Universal Robots PolyScope program: kg_client.urp

Program kg_client (installation=default directory=/home/kieran/ursim-3.12.1.90940/programs createdIn=3.3.4.310 lastSavedIn=3.12.1.90940 robotSerialNumber=2018359999)
Calibrated DH parameters: a=[0.00011, -0.28299, -0.391817, -0.000036, 0.000148, 0]; d=[0.089132, -365.338436, 366.566923, -1.118136, 0.094823, 0.082571]; alpha=[1.570367, -0.000867, -0.014051, 1.570127, -1.570349, 0]; deltaTheta=[0.000049, 0.840298, -0.88576, 0.044111, 0.000904, -0.000211]
BeforeStart
  var_1 := False
  thread_flag := False
  var_10 := [0,0,0,0,0,0,0,0,0,0]
  Set NoAction tcp=TCP
Robot Program (runOnlyOnce=false)
  Loop While (checkContinuously=false) expression=var_1==False
    var_1 := socket_open("127.0.0.1",30010)
    Wait Sleep waitTime=0.5
  Loop While (checkContinuously=true) expression=var_1== True
    Wait Sleep waitTime=0.001
    var_2 := socket_read_ascii_float(12)
    Loop While (checkContinuously=false) expression=var_2[0]≠12
      var_2 := socket_read_ascii_float(12)
    Switch expression=var_2[1]
      Case (caseValue=0)
        'movejl'
        var_3 := p[var_2[2],var_2[3],var_2[4],var_2[5],var_2[6],var_2[7]]
        Script: movej(var_3,var_2[8],var_2[9],var_2[10],var_2[11])
        If var_2[12]==0
          Script: socket_send_string("completed_pose_move")
      Case (caseValue=1)
        'movej'
        var_6 := [var_2[2],var_2[3],var_2[4],var_2[5],var_2[6],var_2[7]]
        Script: movej(var_6,var_2[8],var_2[9],var_2[10],var_2[11])
        If var_2[12]==0
          Script: socket_send_string("completed_joint_move")
      Case (caseValue=2)
        'movel'
        var_3 := p[var_2[2],var_2[3],var_2[4],var_2[5],var_2[6],var_2[7]]
        Script: movel(var_3,var_2[8],var_2[9],var_2[10],var_2[11])
        If var_2[12]==0
          Script: socket_send_string("completed_linear_move")
      Case (caseValue=3)
        'move to var_3 relative to current pose'
        var_3 := p[var_2[2],var_2[3],var_2[4],var_2[5],var_2[6],var_2[7]]
        var_5 := get_actual_tcp_pose()
        Script: movel(pose_trans(var_5,var_3),var_2[8],var_2[9],var_2[10],var_2[11])
        If var_2[12]==0
          Script: socket_send_string("completed_relative_linear_move")
      Case (caseValue=4)
        'force move in single axis'
        var_5 := get_actual_tcp_pose()
        If var_2[2]≠0
          Script: var_5[0]=var_5[0]+var_2[2]
          axis := 0
        ElseIf var_2[3]≠0
          Script: var_5[1]=var_5[1]+var_2[3]
          axis := 1
        ElseIf var_2[4]≠0
          Script: var_5[2]=var_5[2]+var_2[4]
          axis := 2
        Script: thread_flag= True
        Loop While (checkContinuously=true) expression=thread_flag== True
          Script: movel(var_5,var_2[8],var_2[9],0,0)
          Wait Sleep waitTime=0.01
          Script: thread_flag= False
        Script: stopl(10)
        If var_2[12]==0
          Script: socket_send_string("completed_force_move")
      Case (caseValue=5)
        'servoj'
        var_3 := p[var_2[2],var_2[3],var_2[4],var_2[5],var_2[6],var_2[7]]
        If var_2[12]==0
          Script: stopl(0.5)
        Else 
          var_14 := get_inverse_kin(var_3)
          Script: servoj(var_14,t=var_2[9],lookahead_time=var_2[10],gain=var_2[11])
        If var_2[12]==0
          Script: socket_send_string("completed_servoj_move")
      Case (caseValue=6)
        'speedl'
        var_6 := [var_2[2],var_2[3],var_2[4],var_2[5],var_2[6],var_2[7]]
        If var_2[10]==0
          Script: speedl(var_6,var_2[8])
        Else 
          Script: speedl(var_6,var_2[8],var_2[10])
        Script: socket_send_string("completed_speedl")
      Case (caseValue=7)
        'speedj'
        var_6 := [var_2[2],var_2[3],var_2[4],var_2[5],var_2[6],var_2[7]]
        If var_2[10]==0
          Script: speedj(var_6,var_2[8])
        Else 
          Script: speedj(var_6,var_2[8],var_2[10])
        Script: socket_send_string("completed_speedj")
      Case (caseValue=8)
        'stopl'
        Script: stopl(var_2[8])
        Script: socket_send_string("completed_stopl")
      Case (caseValue=9)
        'servoc'
        var_3 := p[var_2[2],var_2[3],var_2[4],var_2[5],var_2[6],var_2[7]]
        If var_2[12]==0
          Script: stopl(var_2[8])
        Else 
          Script: servoc(var_3,a=var_2[8],v=var_2[9],r=var_2[11])
        If var_2[12]==0
          Script: socket_send_string("completed_servoc_move")
      Case (caseValue=10)
        'return current pose'
        var_5 := get_actual_tcp_pose()
        Script: socket_send_string(var_5)
      Case (caseValue=11)
        'return current joints'
        var_4 := get_actual_joint_positions()
        Script: socket_send_string(var_4)
      Case (caseValue=12)
        'return inverse kin of pose'
        var_3 := p[var_2[2],var_2[3],var_2[4],var_2[5],var_2[6],var_2[7]]
        Script: socket_send_string(get_inverse_kin(var_3))
      Case (caseValue=13)
        'return translation to get to 2nd pose from 1st pose coord system'
        var_3 := p[var_2[2],var_2[3],var_2[4],var_2[5],var_2[6],var_2[7]]
        var_5 := get_actual_tcp_pose()
        Script: socket_send_string(pose_trans(var_5,var_3))
      Case (caseValue=14)
        'return current forces'
        Script: socket_send_string(get_tcp_force())
      Case (caseValue=15)
        'return force magnitude'
        Script: socket_send_string(force())
      Case (caseValue=16)
        'return tool velocity'
        Script: socket_send_string(get_actual_tcp_speed())
      Case (caseValue=17)
        'return force magnitude'
        Script: socket_send_string(get_actual_joint_speeds())
      Case (caseValue=20)
        'set tcp'
        var_3 := p[var_2[2],var_2[3],var_2[4],var_2[5],var_2[6],var_2[7]]
        Script: set_tcp(var_3)
        If var_2[12]==0
          Script: socket_send_string("tcp_updated")
      Case (caseValue=21)
        'set payload'
        Script: set_payload(var_2[8],[var_2[2],var_2[3],var_2[4]])
        If var_2[12]==0
          Script: socket_send_string("payload_updated")
      Case (caseValue=22)
        'set digital out'
        If var_2[9]==1
          Script: set_configurable_digital_out(var_2[8], True )
        Else 
          Script: set_configurable_digital_out(var_2[8], False )
        If var_2[12]==0
          Script: socket_send_string("digital output set")
      Case (caseValue=30)
        Script: freedrive_mode()
        Script: socket_send_string("begin_freedrive_mode")
      Case (caseValue=31)
        Script: end_freedrive_mode()
        Script: socket_send_string("end_freedrive_mode")
      Case (caseValue=32)
        Script: socket_send_string("begin_blend_move")
        var_13 := var_2[8]
        n := 0
        Loop While (checkContinuously=false) expression=n<var_13
          Script: n=n+1
          Loop While (checkContinuously=false) expression=var_2[0]≠12
            var_2 := socket_read_ascii_float(12)
          var_3 := p[var_2[2],var_2[3],var_2[4],var_2[5],var_2[6],var_2[7]]
          Script: var_10[n] = var_3
        Script: movel(var_10[0],0.1,0.5,0,0)
        n := 0
        Loop While (checkContinuously=false) expression=n<var_13
          Script: n=n+1
          Script: movep(var_10[n])
      Case (caseValue=33)
        Script: socket_send_string("begin_blend_move")
      Case (caseValue=40)
        Script: socket_send_string("robot_ready")
      Case (caseValue=100)
        'reset program'
        If var_2[12]==0
          Script: socket_send_string("resetting...")
        Script: socket_close()
        var_1 := False
      Case (caseValue=101)
        Script: socket_send_string("ready")
      Case (caseValue=400)
        'safe move'
        var_3 := p[var_2[2],var_2[3],var_2[4],var_2[5],var_2[6],var_2[7]]
        var_5 := get_actual_tcp_pose()
        var_7 := get_inverse_kin(var_3)
        var_8 := get_inverse_kin(var_5)
        var_9 := 0
        Loop Counting (count=6) loopVariable(name=Loop_5)
          If (var_7[Loop_5]-var_8[Loop_5])>2.0  or  (var_8[Loop_5]-var_7[Loop_5])>2.0
            Script: var_9=1
            SuppressedNode
              Script: break
        If var_9==0
          Script: movej(var_3,1,var_2[8],0,0)
          Script: socket_send_string("completed_pose_move")
        Else 
          Script: socket_send_string("no_safe_move_found")
    SuppressedNode
      Wait Sleep waitTime=20
Thread Thread_1 (runOnlyOnce=false)
  Loop While (checkContinuously=false) expression=thread_flag== False
    Script: var_12=0
    Wait Sleep waitTime=0.01
  Wait Sleep waitTime=0.001
  var_11 := get_tcp_force()
  If var_11[axis]*var_11[axis]<var_2[11]*var_2[11]
    Script: var_12=0
  Else 
    Script: var_12=var_12+1
    If var_12>0
      Script: thread_flag= False
      SuppressedNode
        Script: stopl(1)
      SuppressedNode
        Script: speedl([0,0,0,0,0,0],1,0)
